(* PLC project  *)

PROGRAM P
  VAR
    TON_0 : TON;
  END_VAR

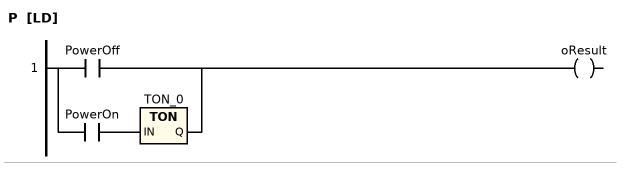
(* LD diagram, written out as Structured Text *)
TON_0(IN := PowerOn);
oResult := PowerOff OR TON_0.Q;
END_PROGRAM
